// TIA Portal V15.1 export
// export: Created 2024-06-21T08:41:14.2414123Z, ExportSetting WithDefaults, DisplayName Totally Integrated Automation Portal, DisplayVersion V15.1 Update 5, DisplayName TIA Portal Openness, DisplayVersion V15.1 Update 5, DisplayName SINAMICS Startdrive Advanced, DisplayVersion V15.1, DisplayName G130, G150, S120, S150, SINAMICS MV, S210, DisplayVersion V15.1, DisplayName G110M, G120, G120C, G120D, G120P, DisplayVersion V15.1, DisplayName STEP 7 Professional, DisplayVersion V15.1 Update 5, DisplayName STEP 7 Safety, DisplayVersion V15.1, DisplayName WinCC Professional, DisplayVersion V15.1 Update 5, DisplayName SIMATIC Visualization Architect, DisplayVersion V15.1
FUNCTION_BLOCK "LGBTrfIn"   // FB6604, FBD
TITLE = LTrfIn / LGBTrfIn
{ S7_Optimized_Access := 'TRUE' }
AUTHOR : VCC
FAMILY : Transpor
VERSION : 0.1
// =============================================================================
// The TrfIn function is a standard FB to be used in all transport functions (as 
// roller, cross-section, …) to execute an IN transfer in automatic Mode or in 
// manual Mode.
// The module will generate the signal O_TrfInCmd to be used by the Motor loop 
// block to steer the Motor.
// It will also generate handshake signals :
// "O_Ready To Receive (Ready to Receive) to inform previous equipement that this 
// equipement is ready to receive a new body,
// "O_Arrived to inform the previous equipment that transfer is done,
// "O_Finish to inform the master sequence that the transport function has 
// finished.
// =============================================================================
// stored: AutoNumber false, IsIECCheckEnabled false, IsRetainMemResEnabled false, MemoryReserve 100, SetENOAutomatically False, UDAEnableTagReadback false
   VAR_INPUT
      I_AnyDet { ExternalAccessible := 'False'; ExternalVisible := 'False'; ExternalWritable := 'False'} : Bool;   // OR of ALL detections / OR of ALL Detections
      I_StopDet { ExternalAccessible := 'False'; ExternalVisible := 'False'; ExternalWritable := 'False'} : Bool;   // Stop detection / Stop Detection
      I_LocalPB { ExternalAccessible := 'False'; ExternalVisible := 'False'; ExternalWritable := 'False'} : Bool;   // Push button (used in manual mode) on local panel / Push button (used in manual Mode) on local panel
      I_ManInfeedAllowed { ExternalAccessible := 'False'; ExternalVisible := 'False'; ExternalWritable := 'False'} : Bool;   // Manual Infeed Allowed (without PushButton)
      I_TrfInBegin { ExternalAccessible := 'False'; ExternalVisible := 'False'; ExternalWritable := 'False'} : Bool;   // Load Begin: condition to start transfer IN
      I_InterlockOk { ExternalAccessible := 'False'; ExternalVisible := 'False'; ExternalWritable := 'False'} : Bool;   // Interlock
      I_ReadyForOperation { ExternalAccessible := 'False'; ExternalVisible := 'False'; ExternalWritable := 'False'} : Bool;   // Ready for operation / Motor Loop Ready for operation
      I_TrfInRdyDlv { ExternalAccessible := 'False'; ExternalVisible := 'False'; ExternalWritable := 'False'} : Bool;   // Ready to deliver: Signal from previous object
      I_TrfInOutfeedHold { ExternalAccessible := 'False'; ExternalVisible := 'False'; ExternalWritable := 'False'} : Bool;   // Outfeed hold in traintransport
      I_TrfInTM { ExternalAccessible := 'False'; ExternalVisible := 'False'; ExternalWritable := 'False'} : Bool;   // Transfer busy signal from previous equipement
      I_TrfOutTM { ExternalAccessible := 'False'; ExternalVisible := 'False'; ExternalWritable := 'False'} : Bool;   // Transfer busy signal to next equipement
      I_ProductionStop { ExternalAccessible := 'False'; ExternalVisible := 'False'; ExternalWritable := 'False'} : Bool;   // ProductionStop from Control Room
      I_TrainCond { ExternalAccessible := 'False'; ExternalVisible := 'False'; ExternalWritable := 'False'} : Bool;   // Train transport used
      I_EnableAlarm { ExternalAccessible := 'False'; ExternalVisible := 'False'; ExternalWritable := 'False'} : Bool := TRUE;   // Enable Alarm
      I_ForcedMan { ExternalAccessible := 'False'; ExternalVisible := 'False'; ExternalWritable := 'False'} : Bool;   // Forced manual
      I_GenRevSw { ExternalAccessible := 'False'; ExternalVisible := 'False'; ExternalWritable := 'False'} : Bool;   // General reverse switch
      I_GeneralPB { ExternalAccessible := 'False'; ExternalVisible := 'False'; ExternalWritable := 'False'} : Bool;   // Push Button is activated in manual (general pushbutton) / Push Button is Activated in manual (general Pushbutton )
   END_VAR
   VAR_OUTPUT
      O_TrfInCmd { ExternalAccessible := 'False'; ExternalVisible := 'False'; ExternalWritable := 'False'} : Bool;   // Command to actuator after interlock / Command to actuator after Interlock
      O_TrfInRdyRcv { ExternalAccessible := 'False'; ExternalVisible := 'False'; ExternalWritable := 'False'} : Bool;   // Ready to Receive: Signal to previous object
      O_TrfInInfeedHold { ExternalAccessible := 'False'; ExternalVisible := 'False'; ExternalWritable := 'False'} : Bool;   // Infeed hold in traintransport
      O_TrfInArrived { ExternalAccessible := 'False'; ExternalVisible := 'False'; ExternalWritable := 'False'} : Bool;   // Body Arrived: Signal to previous object
      O_StopTrfOutCmd { ExternalAccessible := 'False'; ExternalVisible := 'False'; ExternalWritable := 'False'} : Bool;   // Body Arrived: Signal to TrfOut module (reset TrfOutCmd) / Body Arrived: Signal to TrfOut module (Reset TrfOutCmd)
      O_TrfInActive { ExternalAccessible := 'False'; ExternalVisible := 'False'; ExternalWritable := 'False'} : Bool;   // Load active: Signal for sequence -> acknowledge for LoadBegin / Load Active: Signal for sequence -> acknowledge for LoadBegin
      O_TrfInFinished { ExternalAccessible := 'False'; ExternalVisible := 'False'; ExternalWritable := 'False'} : Bool;   // Load finished: Signal for sequence -> Load finished
      O_InterlockAlarm { ExternalAccessible := 'False'; ExternalVisible := 'False'; ExternalWritable := 'False'} : Bool;   // Interlock alarm (0=No alarm/1=Alarm) / Interlock Alarm (0=No Alarm/1=Alarm)
   END_VAR
   VAR_IN_OUT
      IO_Modes : "Modes";   // Modes
      H_HMI : "H_HMI";   // Animation
      H_TrfIn : "H_TrfIn";   // Animation
      H_FncSelInHMI { ExternalAccessible := 'False'; ExternalVisible := 'False'; ExternalWritable := 'False'} : Bool;   // This function is selected to run from HMI / This function is Selected to run from HMI
      C_TrfInUsed { ExternalAccessible := 'False'; ExternalVisible := 'False'; ExternalWritable := 'False'} : Bool;   // This FB is used
   END_VAR
   VAR RETAIN
      TrfInCmdRequest { ExternalAccessible := 'False'; ExternalVisible := 'False'; ExternalWritable := 'False'} : Bool;   // Command request before interlock / Command Request before Interlock
      BeenLowStopDet { ExternalAccessible := 'False'; ExternalVisible := 'False'; ExternalWritable := 'False'} : Bool;   // Memory that StopDet has been low
      StopDetOffDelayed { ExternalAccessible := 'False'; ExternalVisible := 'False'; ExternalWritable := 'False'} : Bool;   // Memory that StopDet has been low + timer
      TrfInOkToBeginAutoMc { ExternalAccessible := 'False'; ExternalVisible := 'False'; ExternalWritable := 'False'} : Bool;   // AutoMem Ready to Receive: Signal to previous object
      TrfInCmd { ExternalAccessible := 'False'; ExternalVisible := 'False'; ExternalWritable := 'False'} : Bool;   // MEM Command to actuator after interlock / Command to actuator after Interlock
      TrfInRdyRcv { ExternalAccessible := 'False'; ExternalVisible := 'False'; ExternalWritable := 'False'} : Bool;   // MEM Ready to Receive: Signal to previous object / Ready to Receive: Signal to previous object
      TrfInArrived { ExternalAccessible := 'False'; ExternalVisible := 'False'; ExternalWritable := 'False'} : Bool;   // MEM Arrived signal / Arrived signal
      StopTrfOutCmd { ExternalAccessible := 'False'; ExternalVisible := 'False'; ExternalWritable := 'False'} : Bool;   // MEM Arrived signal to TrfOut (reset TrfOutCmd) / Arrived signal to TrfOut (Reset TrfOutCmd)
      InterlockAlarm { ExternalAccessible := 'False'; ExternalVisible := 'False'; ExternalWritable := 'False'} : Bool;   // MEM Interlock alarm / Interlock Alarm
      TrfInFinished { ExternalAccessible := 'False'; ExternalVisible := 'False'; ExternalWritable := 'False'} : Bool;   // Load finished: Signal for sequence -> Load finished
   END_VAR
   VAR
      TimerBeenLowStpDet { ExternalAccessible := 'False'; ExternalVisible := 'False'; ExternalWritable := 'False'} : "LTimer";   // FB
      TOF_TrfInFinished { ExternalAccessible := 'False'; ExternalVisible := 'False'; ExternalWritable := 'False'} : TOF_TIME;
      TOF_TrfInArrived { ExternalAccessible := 'False'; ExternalVisible := 'False'; ExternalWritable := 'False'} : TOF_TIME;
   END_VAR
   VAR_TEMP   // added for the SCL form of the ladder/FBD networks
      _w1 : Bool;
   END_VAR
BEGIN

REGION Network 1: **** 1 - Inputs **** Memory of BeenLowDetStop
   // Memory of BeenLowDetStop
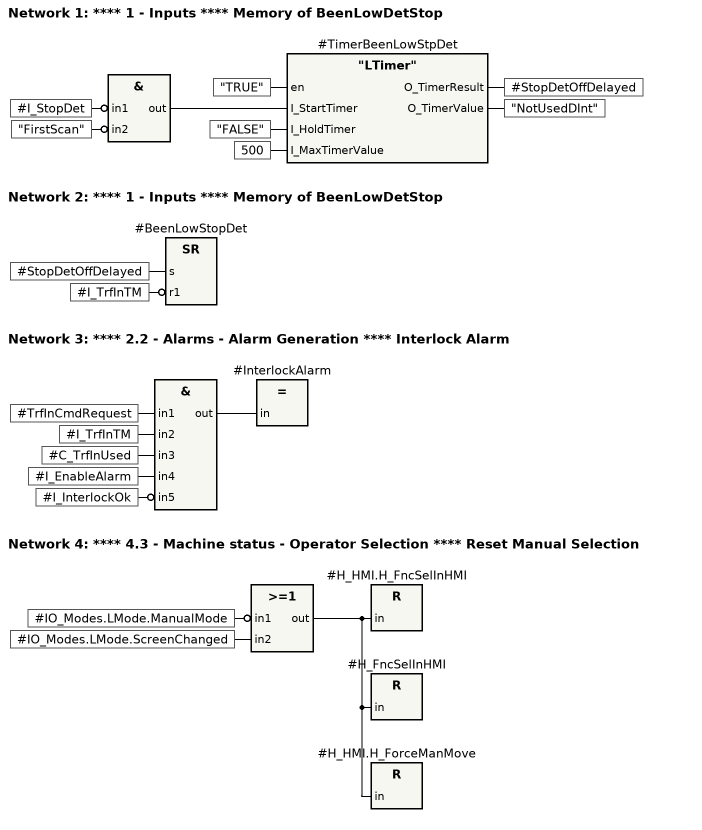
   IF "TRUE" THEN
       #TimerBeenLowStpDet(I_StartTimer := NOT #I_StopDet AND NOT "FirstScan",   // "LTimer"
                           I_HoldTimer := "FALSE",
                           I_MaxTimerValue := 500,
                           O_TimerResult => #StopDetOffDelayed,
                           O_TimerValue => "NotUsedDInt");
   END_IF;
END_REGION

REGION Network 2: **** 1 - Inputs **** Memory of BeenLowDetStop
   // Memory of BeenLowDetStop
   IF #StopDetOffDelayed THEN
       #BeenLowStopDet := TRUE;   // SR flip-flop
   END_IF;
   IF NOT #I_TrfInTM THEN #BeenLowStopDet := FALSE; END_IF;
END_REGION

REGION Network 3: **** 2.2 - Alarms - Alarm Generation **** Interlock Alarm
   // Interlock Alarm
   #InterlockAlarm := #TrfInCmdRequest AND #I_TrfInTM AND #C_TrfInUsed AND #I_EnableAlarm AND NOT #I_InterlockOk;
END_REGION

REGION Network 4: **** 4.3 - Machine status - Operator Selection **** Reset Manual Selection
   // Reset Manual Selection
   IF NOT #IO_Modes.LMode.ManualMode OR #IO_Modes.LMode.ScreenChanged THEN
       #H_HMI.H_FncSelInHMI := FALSE;
       #H_FncSelInHMI := FALSE;
       #H_HMI.H_ForceManMove := FALSE;
   END_IF;
END_REGION

REGION Network 5: **** 4.6 - Machine Status - Indication **** Icon Animation
   // Icon Animation
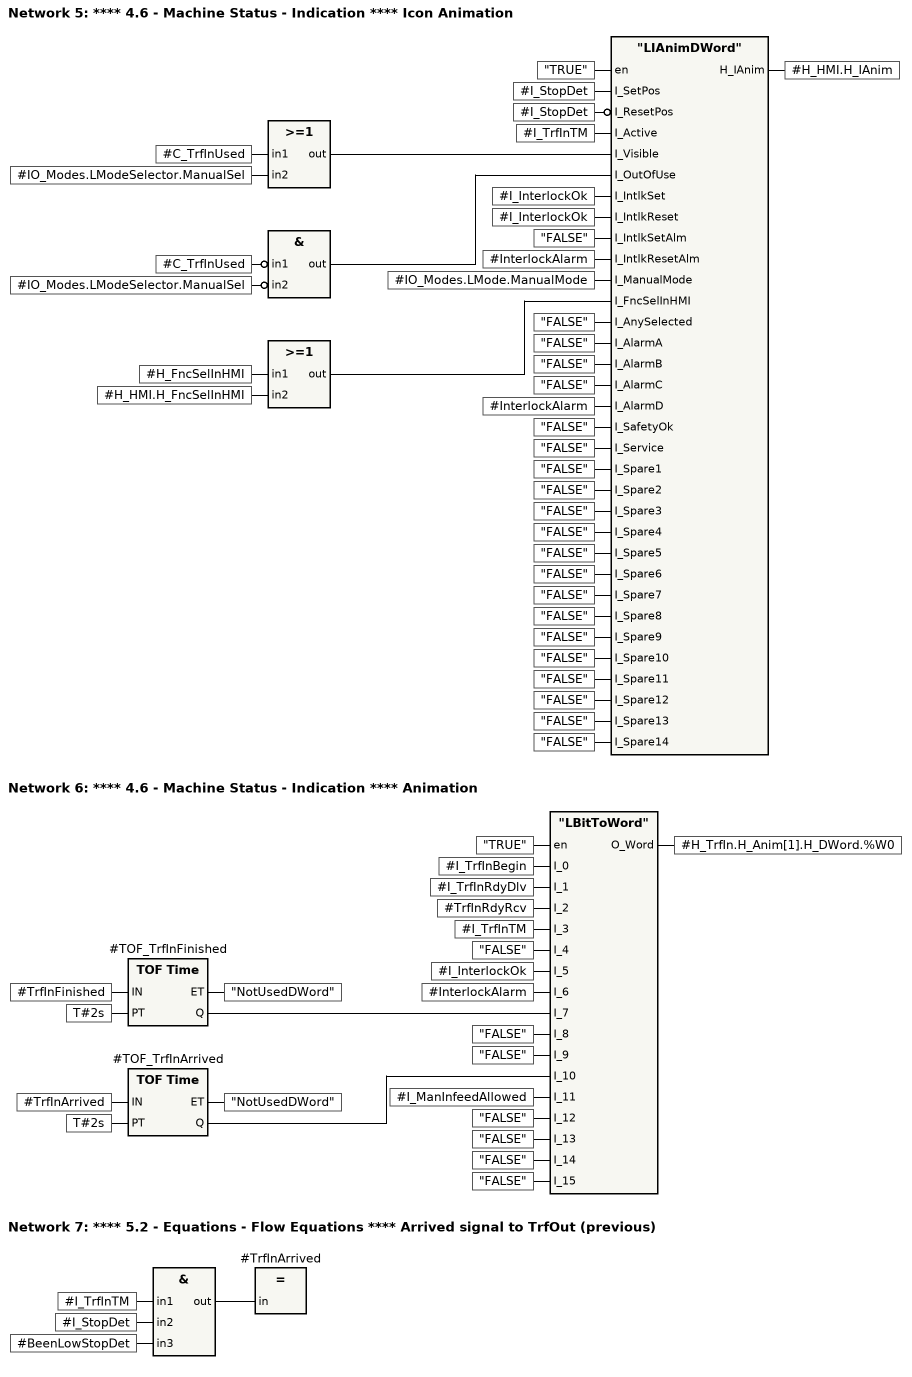
   IF "TRUE" THEN
       "LIAnimDWord"(I_SetPos := #I_StopDet,
                     I_ResetPos := NOT #I_StopDet,
                     I_Active := #I_TrfInTM,
                     I_Visible := #C_TrfInUsed OR #IO_Modes.LModeSelector.ManualSel,
                     I_OutOfUse := NOT #C_TrfInUsed AND NOT #IO_Modes.LModeSelector.ManualSel,
                     I_IntlkSet := #I_InterlockOk,
                     I_IntlkReset := #I_InterlockOk,
                     I_IntlkSetAlm := "FALSE",
                     I_IntlkResetAlm := #InterlockAlarm,
                     I_ManualMode := #IO_Modes.LMode.ManualMode,
                     I_FncSelInHMI := #H_FncSelInHMI OR #H_HMI.H_FncSelInHMI,
                     I_AnySelected := "FALSE",
                     I_AlarmA := "FALSE",
                     I_AlarmB := "FALSE",
                     I_AlarmC := "FALSE",
                     I_AlarmD := #InterlockAlarm,
                     I_SafetyOk := "FALSE",
                     I_Service := "FALSE",
                     I_Spare1 := "FALSE",
                     I_Spare2 := "FALSE",
                     I_Spare3 := "FALSE",
                     I_Spare4 := "FALSE",
                     I_Spare5 := "FALSE",
                     I_Spare6 := "FALSE",
                     I_Spare7 := "FALSE",
                     I_Spare8 := "FALSE",
                     I_Spare9 := "FALSE",
                     I_Spare10 := "FALSE",
                     I_Spare11 := "FALSE",
                     I_Spare12 := "FALSE",
                     I_Spare13 := "FALSE",
                     I_Spare14 := "FALSE",
                     H_IAnim => #H_HMI.H_IAnim);
   END_IF;
END_REGION

REGION Network 6: **** 4.6 - Machine Status - Indication **** Animation
   // Animation
   #TOF_TrfInFinished(IN := #TrfInFinished, PT := T#2s, ET => "NotUsedDWord");   // TOF
   #TOF_TrfInArrived(IN := #TrfInArrived, PT := T#2s, ET => "NotUsedDWord");   // TOF
   IF "TRUE" THEN
       "LBitToWord"(I_0 := #I_TrfInBegin,
                    I_1 := #I_TrfInRdyDlv,
                    I_2 := #TrfInRdyRcv,
                    I_3 := #I_TrfInTM,
                    I_4 := "FALSE",
                    I_5 := #I_InterlockOk,
                    I_6 := #InterlockAlarm,
                    I_7 := #TOF_TrfInFinished.Q,
                    I_8 := "FALSE",
                    I_9 := "FALSE",
                    I_10 := #TOF_TrfInArrived.Q,
                    I_11 := #I_ManInfeedAllowed,
                    I_12 := "FALSE",
                    I_13 := "FALSE",
                    I_14 := "FALSE",
                    I_15 := "FALSE",
                    O_Word => #H_TrfIn.H_Anim[1].H_DWord.%W0);
   END_IF;
END_REGION

REGION Network 7: **** 5.2 - Equations - Flow Equations **** Arrived signal to TrfOut (previous)
   // Arrived signal to TrfOut (previous)
   #TrfInArrived := #I_TrfInTM AND #I_StopDet AND #BeenLowStopDet;
END_REGION

REGION Network 8: **** 5.2 - Equations - Flow Equations **** Arrived signal to TrfOut in the same roller to stop the Motor command.
   // Arrived signal to TrfOut in the same roller to stop the Motor command. Only 
   // needed for train transport when theis transport is finished before the next 
   // transport.
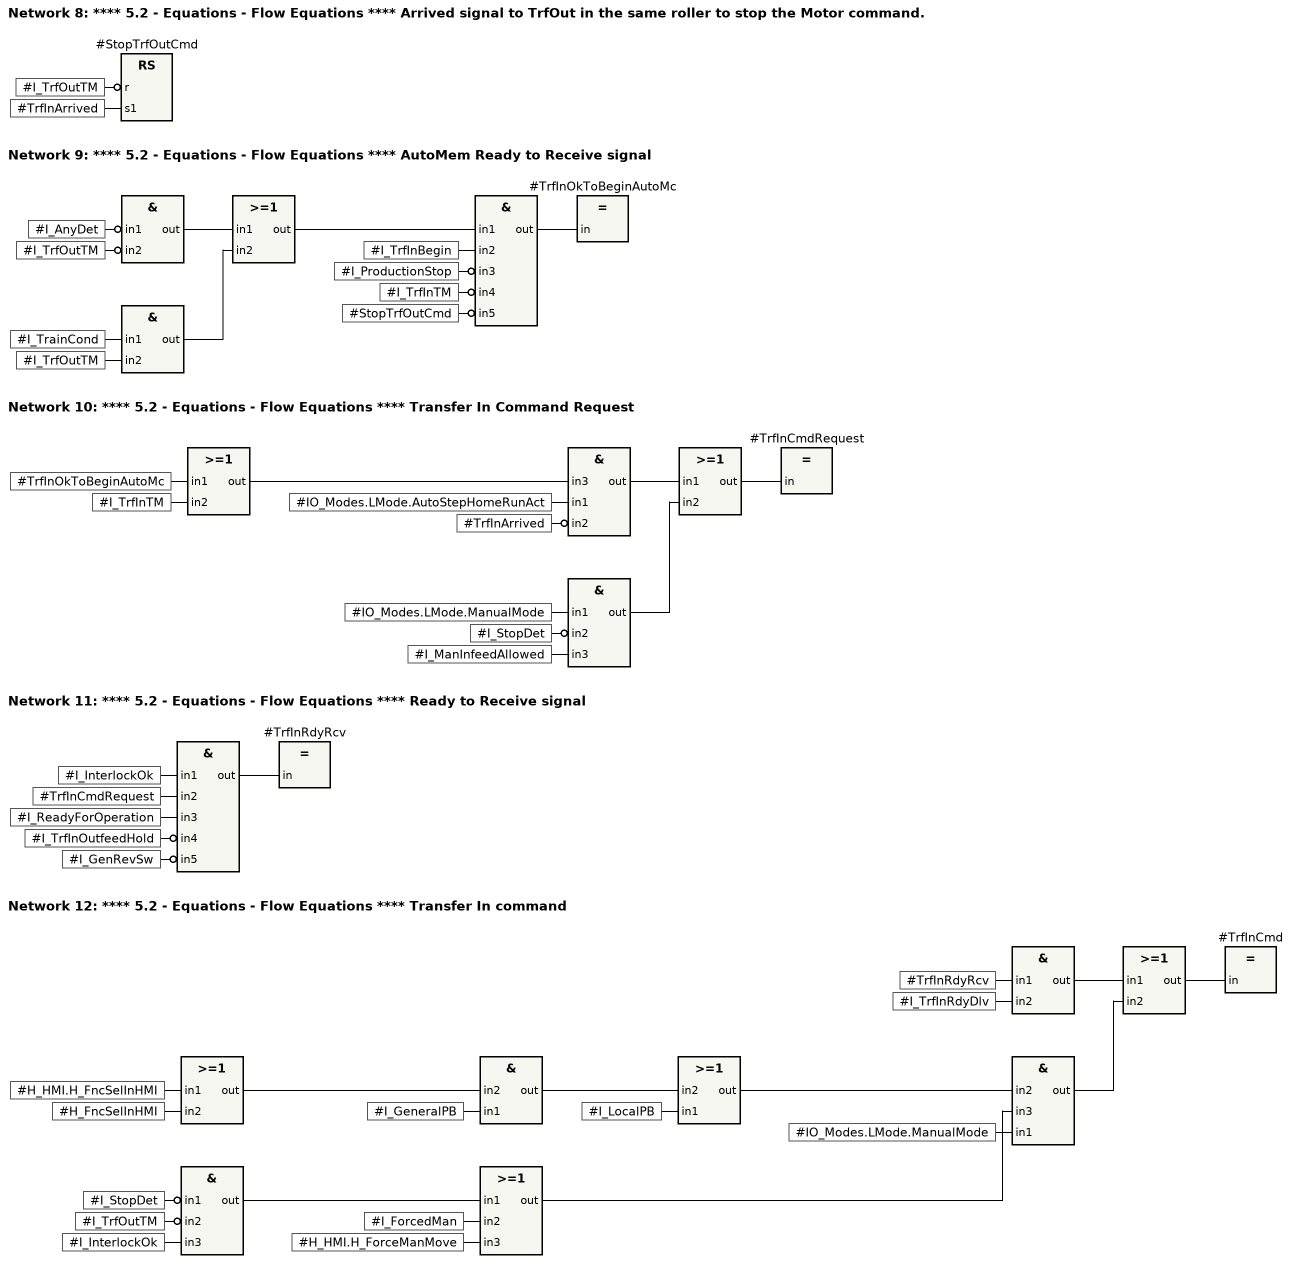
   IF NOT #I_TrfOutTM THEN
       #StopTrfOutCmd := FALSE;   // RS flip-flop
   END_IF;
   IF #TrfInArrived THEN #StopTrfOutCmd := TRUE; END_IF;
END_REGION

REGION Network 9: **** 5.2 - Equations - Flow Equations **** AutoMem Ready to Receive signal
   // AutoMem Ready to Receive signal
   #TrfInOkToBeginAutoMc := ((NOT #I_AnyDet AND NOT #I_TrfOutTM) OR (#I_TrainCond AND #I_TrfOutTM)) AND #I_TrfInBegin AND NOT #I_ProductionStop AND NOT #I_TrfInTM AND NOT #StopTrfOutCmd;
END_REGION

REGION Network 10: **** 5.2 - Equations - Flow Equations **** Transfer In Command Request
   // Transfer In Command Request
   #TrfInCmdRequest := ((#TrfInOkToBeginAutoMc OR #I_TrfInTM) AND #IO_Modes.LMode.AutoStepHomeRunAct AND NOT #TrfInArrived) OR (#IO_Modes.LMode.ManualMode AND NOT #I_StopDet AND #I_ManInfeedAllowed);
END_REGION

REGION Network 11: **** 5.2 - Equations - Flow Equations **** Ready to Receive signal
   // Ready to Receive signal
   #TrfInRdyRcv := #I_InterlockOk AND #TrfInCmdRequest AND #I_ReadyForOperation AND NOT #I_TrfInOutfeedHold AND NOT #I_GenRevSw;
END_REGION

REGION Network 12: **** 5.2 - Equations - Flow Equations **** Transfer In command
   // Transfer In command
   // 1. Automatic Ready To Receive and Ready To Deliver
   // 2. Manual from HMI and general setPB or via local panel
   #TrfInCmd := (#TrfInRdyRcv AND #I_TrfInRdyDlv) OR ((((#H_HMI.H_FncSelInHMI OR #H_FncSelInHMI) AND #I_GeneralPB) OR #I_LocalPB) AND ((NOT #I_StopDet AND NOT #I_TrfOutTM AND #I_InterlockOk) OR #I_ForcedMan OR #H_HMI.H_ForceManMove) AND #IO_Modes.LMode.ManualMode);
END_REGION

REGION Network 13: **** 5.2 - Equations - Flow Equations **** TransferIn InfeedHold
   // TransferIn InfeedHold
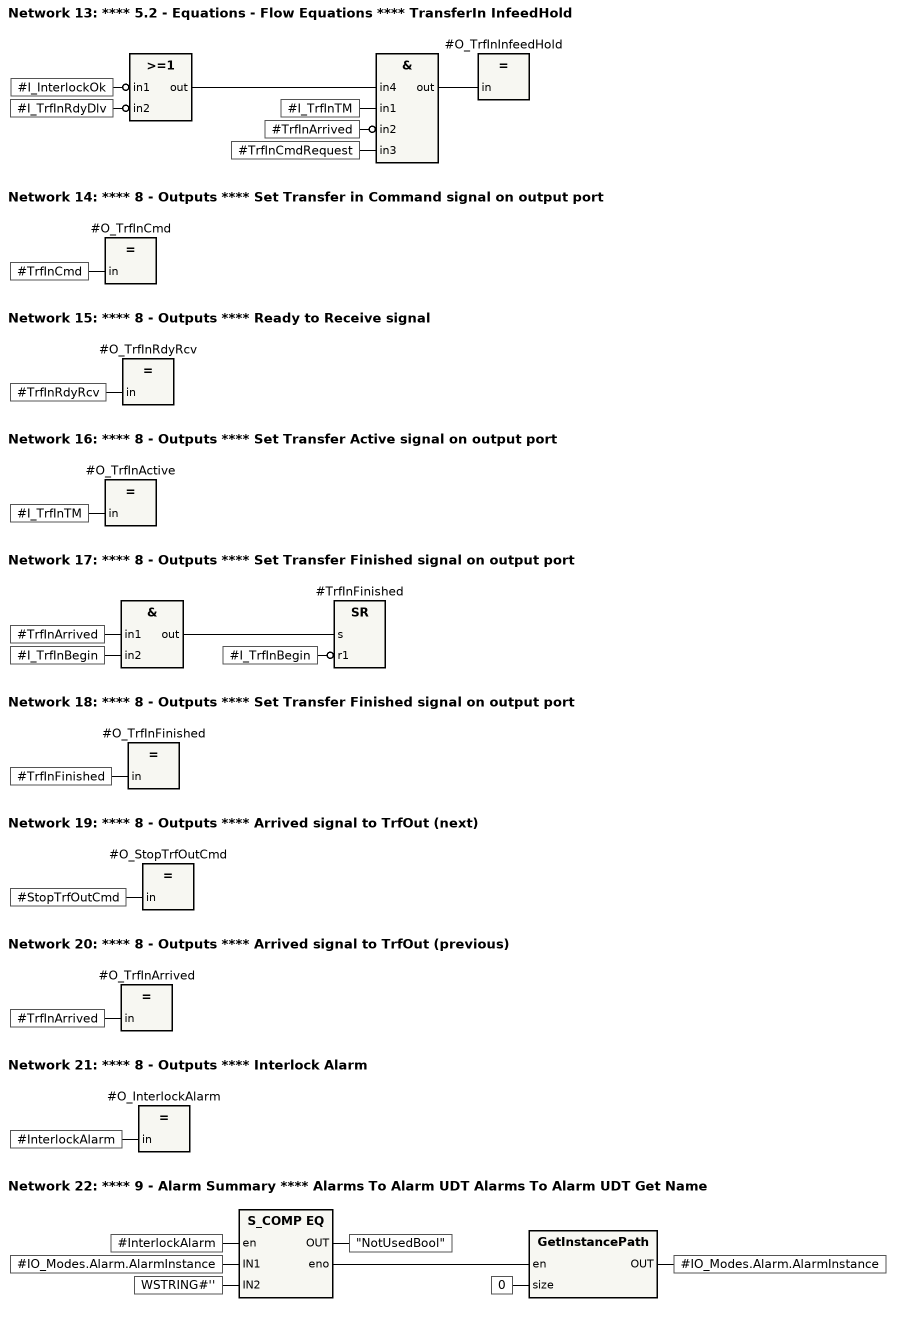
   #O_TrfInInfeedHold := (NOT #I_InterlockOk OR NOT #I_TrfInRdyDlv) AND #I_TrfInTM AND NOT #TrfInArrived AND #TrfInCmdRequest;
END_REGION

REGION Network 14: **** 8 - Outputs **** Set Transfer in Command signal on output port
   // Set Transfer in Command signal on output port
   #O_TrfInCmd := #TrfInCmd;
END_REGION

REGION Network 15: **** 8 - Outputs **** Ready to Receive signal
   // Ready to Receive signal
   #O_TrfInRdyRcv := #TrfInRdyRcv;
END_REGION

REGION Network 16: **** 8 - Outputs **** Set Transfer Active signal on output port
   // Set Transfer Active signal on output port
   #O_TrfInActive := #I_TrfInTM;
END_REGION

REGION Network 17: **** 8 - Outputs **** Set Transfer Finished signal on output port
   // Set Transfer Finished signal on output port
   IF #TrfInArrived AND #I_TrfInBegin THEN
       #TrfInFinished := TRUE;   // SR flip-flop
   END_IF;
   IF NOT #I_TrfInBegin THEN #TrfInFinished := FALSE; END_IF;
END_REGION

REGION Network 18: **** 8 - Outputs **** Set Transfer Finished signal on output port
   // Set Transfer Finished signal on output port
   #O_TrfInFinished := #TrfInFinished;
END_REGION

REGION Network 19: **** 8 - Outputs **** Arrived signal to TrfOut (next)
   // Arrived signal to TrfOut (next)
   #O_StopTrfOutCmd := #StopTrfOutCmd;
END_REGION

REGION Network 20: **** 8 - Outputs **** Arrived signal to TrfOut (previous)
   // Arrived signal to TrfOut (previous)
   #O_TrfInArrived := #TrfInArrived;
END_REGION

REGION Network 21: **** 8 - Outputs **** Interlock Alarm
   // Interlock Alarm
   #O_InterlockAlarm := #InterlockAlarm;
END_REGION

REGION Network 22: **** 9 - Alarm Summary **** Alarms To Alarm UDT Alarms To Alarm UDT Get Name
   // Alarm / Alarm D
   S_COMP(EN := #InterlockAlarm,
          IN1 := #IO_Modes.Alarm.AlarmInstance,
          IN2 := WSTRING#'',
          OUT => "NotUsedBool",
          ENO => #_w1);
   IF #_w1 THEN GetInstancePath(size := 0, OUT => #IO_Modes.Alarm.AlarmInstance); END_IF;
END_REGION

REGION Network 23: **** 9 - Alarm Summary **** Alarms To Alarm UDT
   // Alarm / Alarm D
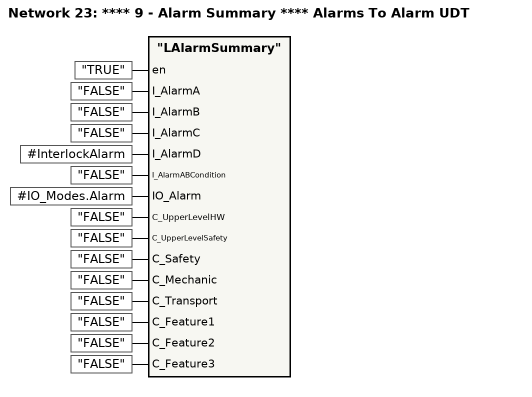
   IF "TRUE" THEN
       "LAlarmSummary"(I_AlarmA := "FALSE",
                       I_AlarmB := "FALSE",
                       I_AlarmC := "FALSE",
                       I_AlarmD := #InterlockAlarm,
                       I_AlarmABCondition := "FALSE",
                       IO_Alarm := #IO_Modes.Alarm,
                       C_UpperLevelHW := "FALSE",
                       C_UpperLevelSafety := "FALSE",
                       C_Safety := "FALSE",
                       C_Mechanic := "FALSE",
                       C_Transport := "FALSE",
                       C_Feature1 := "FALSE",
                       C_Feature2 := "FALSE",
                       C_Feature3 := "FALSE");
   END_IF;
END_REGION
END_FUNCTION_BLOCK
